(*
SPDX-FileCopyrightText: © 2026 Oleksandr Tiutyk <trofimich@gmail.com>
SPDX-License-Identifier: MIT
License: https://opensource.org/license/mit
*)

TYPE HMI_INTERSECTION_CONTROLLER_STATUSES :
STRUCT
	Mode : INTERSECTION_MODE;
	ModeName : STRING(20);
	
	LightsState : INTERSECTION_LIGHTS_STATE;
	LightsStateName : STRING(20);
	
	SwitchingSpeedCorrectionPercent : SINT(-20..+20);
END_STRUCT
END_TYPE

(* stored: Version 1.1.0.1
   DUT HMI_INTERSECTION_CONTROLLER_STATUSES: Id {a9732ba8-50c0-4b74-928a-dacec452f7d1} *)
